Fanuc KAREL source: ko00027.KL

-- PROVISIONAL review KL for V940-1; original PC SHA256 a96047cd7f611757376575bf8bcf7670c1e1e66530b592041bd113ae4569bed7
-- Incomplete behavior may be omitted. Consult companion uncertainty JSON. Do not deploy.
PROGRAM KO00027
%NOLOCKGROUP
-- UNRESOLVED_DECL P1 type=000199
-- UNRESOLVED_DECL P2 type=000199
-- UNRESOLVED_DECL P3 type=000199
-- UNRESOLVED_DECL OUT type=000106
BEGIN
  -- V9_ZERO_TABLE_METADATA_HINT layout=0001; no indexed target words; source/name/runtime held
  -- UNRESOLVED_PC offsets 5-65; opcodes 27,27,49,7E,AD,27,49,7E,AD,27,49,7E,AD,76,7E,4A
  -- UNRESOLVED_PC offsets 70-74; opcodes 7F
END KO00027
